PROGRAM MAIN
VAR
END_VAR

END_PROGRAM

(* stored: Version 1.1.0.1
   POU MAIN: Id {d1ec5373-a180-4b19-a616-98d63a72bfd5} *)
